// TIA Portal V20 export
TYPE "LWONIK_typeFromSafetyDoorStatus"
// stored: Access Published
   STRUCT
      FdoorSwitchStatus : Struct
         UnwinderTopDoorOpen : Bool;
         UnwinderLeftDoorOpen : Bool;
         UnwinderRightDoorOpen : Bool;
         CutterDoorOpen : Bool;
         MagazineDoorOpen : Bool;
         ConveyorDoorOpen : Bool;
         ScrapBoxDoorOpen : Bool;
         ScrapBoxDoorClose : Bool;
         CentralAisleDoorOpen : Bool;
         TotalOneDoorOpen : Bool;
      END_STRUCT;
      FdoorCoilStatus : Struct
         UnwinderTopDoorUnlock : Bool;
         UnwinderLeftDoorUnlock : Bool;
         UnwinderRightDoorUnlock : Bool;
         CutterDoorUnlock : Bool;
         MagazineDoorUnlock : Bool;
         ConveyorDoorUnlock : Bool;
         ScrapBoxDoorUnlock : Bool;
         CentralAisleDoorUnlock : Bool;
         TotalOneDoorUnlock : Bool;
      END_STRUCT;
   END_STRUCT;
END_TYPE
